// TIA Portal project "MATKAP" (V15.1)

(* hardware
DEVICE "S7300/ET200M station_1"  S7-300 station
   slot 0: "Rail_0"  Rail  6ES7 390-1***0-0AA0
   slot 2: "PLC_1"  CPU 314C-2 PN/DP  6ES7 314-6EH04-0AB0  V3.3
      slot 2: "PROFINET interface_1"  PN-IO
         slot 1: "Port_1"  Port
         slot 2: "Port_2"  Port
      slot 5: "DI 24/DO 16_1"  DI24/DO16
      slot 6: "AI 5/AO 2_1"  AI5/AO2
      slot 7: "Count_1"  Counter
      slot 8: "Positioning_1"  Positioning
*)

// ===== PLC "PLC_1"  CPU 314C-2 PN/DP =====

VAR_GLOBAL   // PLC tag table "Default tag table"
   "START" AT %I0.0 : Bool;
   "LAMBA" AT %Q0.0 : Bool;
   "STOP" AT %I0.1 : Bool;
   "L" AT %I0.2 : Bool;
   "M1" AT %Q0.1 : Bool;
   "H" AT %I0.3 : Bool;
   "M2" AT %Q0.2 : Bool;
   "L1" AT %I0.4 : Bool;
   "H1" AT %I0.5 : Bool;
   "Tag_1" AT %M0.0 : Bool;
   "Tag_2" AT %M1.0 : Bool;
   "Tag_3" AT %M0.1 : Bool;
   "Tag_4" AT %M1.1 : Bool;
   "Tag_5" AT %I0.7 : Bool;
   "Tag_6" AT %MW1 : Int;
   "Tag_7" AT %M0.2 : Bool;
   "Tag_8" AT %M1.2 : Bool;
   "Tag_9" AT %M0.3 : Bool;
   "Tag_10" AT %M1.3 : Bool;
END_VAR

ORGANIZATION_BLOCK "Main"   // OB1, LAD
TITLE = "Main Program Sweep (Cycle)"
{ S7_Optimized_Access := 'FALSE' }
VERSION : 0.1
   VAR_TEMP
      OB1_EV_CLASS : Byte;   // Bits 0-3 = 1 (Coming event), Bits 4-7 = 1 (Event class 1)
      OB1_SCAN_1 : Byte;   // 1 (Cold restart scan 1 of OB 1), 3 (Scan 2-n of OB 1)
      OB1_PRIORITY : Byte;   // Priority of OB Execution
      OB1_OB_NUMBR : Byte;   // 1 (Organization block 1, OB1)
      OB1_RESERVED_1 : Byte;   // Reserved for system
      OB1_RESERVED_2 : Byte;   // Reserved for system
      OB1_PREV_CYCLE : Int;   // Cycle time of previous OB1 scan (milliseconds)
      OB1_MIN_CYCLE : Int;   // Minimum cycle time of OB1 (milliseconds)
      OB1_MAX_CYCLE : Int;   // Maximum cycle time of OB1 (milliseconds)
      OB1_DATE_TIME : Date_And_Time;   // Date and time OB1 started
   END_VAR
   VAR_TEMP   // added for the SCL form of the ladder/FBD networks
      _w1 : Bool;
   END_VAR
BEGIN

REGION Network 1
   // START
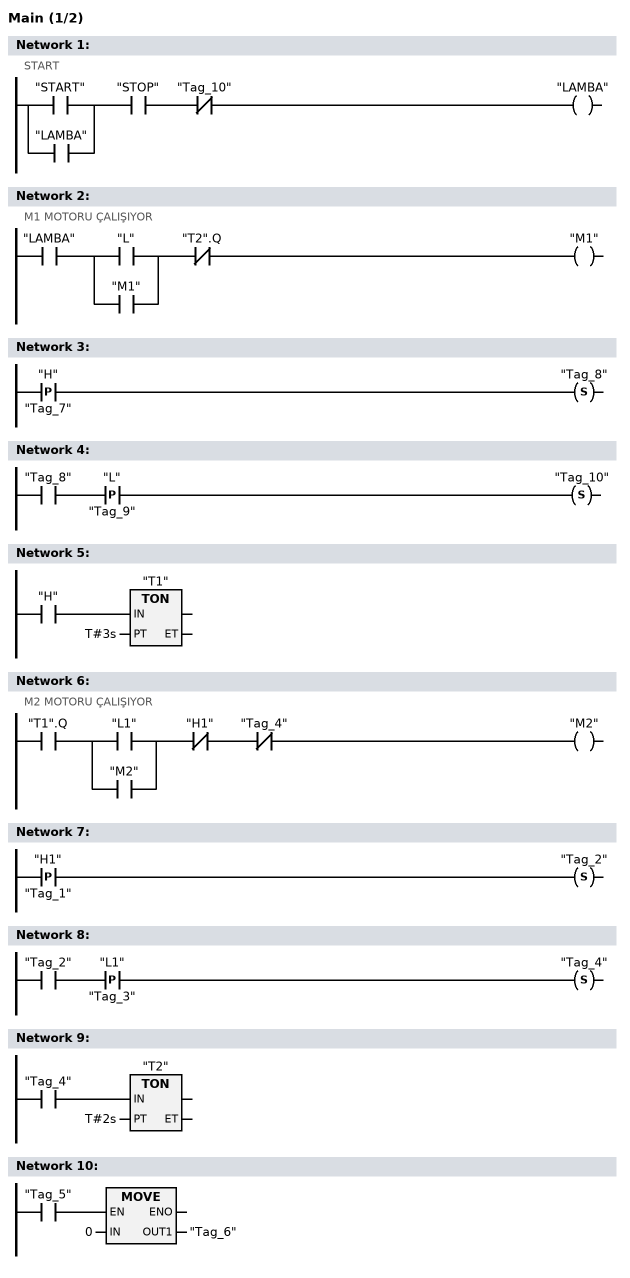
   RUNG wire#powerrail
      Contact( "START" )
      wire#w1
      Contact( "STOP" )
      I_Contact( "Tag_10" )
      Coil( "LAMBA" )
   END_RUNG
   RUNG wire#powerrail
      Contact( "LAMBA" )
   END_RUNG wire#w1
   // the same network as SCL:
   "LAMBA" := ("START" OR "LAMBA") AND "STOP" AND NOT "Tag_10";
END_REGION

REGION Network 2
   // M1 MOTORU ÇALIŞIYOR
   RUNG wire#powerrail
      Contact( "LAMBA" )
      wire#w1
      Contact( "L" )
      wire#w2
      I_Contact( "T2".Q )
      Coil( "M1" )
   END_RUNG
   RUNG wire#w1
      Contact( "M1" )
   END_RUNG wire#w2
   // the same network as SCL:
   "M1" := "LAMBA" AND ("L" OR "M1") AND NOT "T2".Q;
END_REGION

REGION Network 3
   RUNG wire#powerrail
      P_Contact(operand := "H", bit := "Tag_7")
      S_Coil( "Tag_8" )
   END_RUNG
   // the same network as SCL:
   #_w1 := "H" AND NOT "Tag_7";   // rising edge of "H"
   "Tag_7" := "H";
   IF #_w1 THEN "Tag_8" := TRUE; END_IF;
END_REGION

REGION Network 4
   RUNG wire#powerrail
      Contact( "Tag_8" )
      P_Contact(operand := "L", bit := "Tag_9")
      S_Coil( "Tag_10" )
   END_RUNG
   // the same network as SCL:
   #_w1 := "Tag_8" AND "L" AND NOT "Tag_9";   // rising edge of "L"
   "Tag_9" := "L";
   IF #_w1 THEN "Tag_10" := TRUE; END_IF;
END_REGION

REGION Network 5
   "T1".TON(IN := "H", PT := T#3s);
END_REGION

REGION Network 6
   // M2 MOTORU ÇALIŞIYOR
   RUNG wire#powerrail
      Contact( "T1".Q )
      wire#w1
      Contact( "L1" )
      wire#w2
      I_Contact( "H1" )
      I_Contact( "Tag_4" )
      Coil( "M2" )
   END_RUNG
   RUNG wire#w1
      Contact( "M2" )
   END_RUNG wire#w2
   // the same network as SCL:
   "M2" := "T1".Q AND ("L1" OR "M2") AND NOT "H1" AND NOT "Tag_4";
END_REGION

REGION Network 7
   RUNG wire#powerrail
      P_Contact(operand := "H1", bit := "Tag_1")
      S_Coil( "Tag_2" )
   END_RUNG
   // the same network as SCL:
   #_w1 := "H1" AND NOT "Tag_1";   // rising edge of "H1"
   "Tag_1" := "H1";
   IF #_w1 THEN "Tag_2" := TRUE; END_IF;
END_REGION

REGION Network 8
   RUNG wire#powerrail
      Contact( "Tag_2" )
      P_Contact(operand := "L1", bit := "Tag_3")
      S_Coil( "Tag_4" )
   END_RUNG
   // the same network as SCL:
   #_w1 := "Tag_2" AND "L1" AND NOT "Tag_3";   // rising edge of "L1"
   "Tag_3" := "L1";
   IF #_w1 THEN "Tag_4" := TRUE; END_IF;
END_REGION

REGION Network 9
   "T2".TON(IN := "Tag_4", PT := T#2s);
END_REGION

REGION Network 10
   RUNG wire#powerrail
      Contact( "Tag_5" )
      { S7_GenerateENO := "TRUE" } Move(in := 0, out1 => "Tag_6")
   END_RUNG
   // the same network as SCL:
   IF "Tag_5" THEN "Tag_6" := 0; END_IF;
END_REGION

REGION Network 11
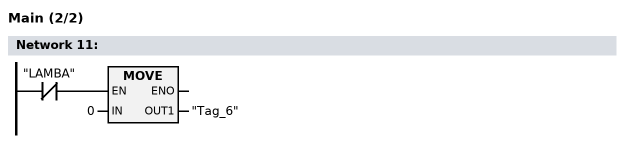
   RUNG wire#powerrail
      I_Contact( "LAMBA" )
      { S7_GenerateENO := "TRUE" } Move(in := 0, out1 => "Tag_6")
   END_RUNG
   // the same network as SCL:
   IF NOT "LAMBA" THEN "Tag_6" := 0; END_IF;
END_REGION
END_ORGANIZATION_BLOCK